INTERFACE I_MotorControl

METHOD GetActualSpeed : INT
END_METHOD

PROPERTY RemoteLocalStatus : bool
GET
END_GET
END_PROPERTY

METHOD SetSpeed : BOOL
VAR_INPUT
	nSetSpeed: INT;
END_VAR
END_METHOD

METHOD StartMotor : BOOL
VAR_INPUT
	bStart: BOOL;
END_VAR
END_METHOD

METHOD StopMotor : BOOL
VAR_INPUT
	bStop: BOOL;
END_VAR
END_METHOD

END_INTERFACE

(* stored: Version 1.1.0.1, ProductVersion 3.1.4024.5
   Itf I_MotorControl: Id {00246e69-092b-4f13-aa0e-aa240ec05aee}
   Method GetActualSpeed: Id {7060f2c1-bf03-4dae-b16d-7ecf37b72c60}
   Property RemoteLocalStatus: Id {d66a6511-d60d-4cae-bd69-eafbd24061c0}
   Get Get: Id {162cefcc-4ad9-41cb-8a7c-b4cb2d066adb}
   Method SetSpeed: Id {0e8b0826-04e5-4db3-b2c3-fd799dee1c6e}
   Method StartMotor: Id {f090f8da-72e2-4947-b461-1a25b85bdf19}
   Method StopMotor: Id {6bc74f6d-1d85-4170-bb81-b7815def02ed} *)
